INTERFACE ICyclic EXTENDS __SYSTEM.IQueryInterface

METHOD Cyclic : BOOL
VAR_INPUT
END_VAR
END_METHOD

END_INTERFACE

(* stored: Version 1.1.0.1
   Itf ICyclic: Id {43fdc5ae-18e4-0595-27b8-5b5f9eaccff3}
   Method Cyclic: Id {979f0ea9-4275-0ecf-15cc-6c54012aa8e2} *)
